FUNCTION_BLOCK FB_LinearMovementWithFeedback
VAR_INPUT
	ToPosition: BOOL;	// TRUE: Moves the drive to position
	Feedback:	BOOL;	// Feedback signal (e.g. reed contact)
	Lock: 		BOOL;	// Interlock for the output
	HoldOutput: BOOL;	// TRUE: Actor remains true when target position reached
END_VAR
VAR_OUTPUT
	Actor:		BOOL;	
END_VAR
VAR
END_VAR

Actor := ToPosition AND NOT Lock AND (HoldOutput OR NOT Feedback);

END_FUNCTION_BLOCK

(* stored: Version 1.1.0.1, ProductVersion 3.1.4024.11
   POU FB_LinearMovementWithFeedback: Id {e55efb08-7dc4-491e-8517-ba928e9c9bd6}, SpecialFunc None *)
